(* PLC project Unnamed, Unknown Unnamed 1 *)
(* stored: creationDateTime 2021-10-03T01:48:44, modificationDateTime 2021-10-03T03:04:46 *)

PROGRAM part2
  VAR
    pos_x0 AT %IX0.0 : BOOL;
    pos_x1 AT %IX0.1 : BOOL;
    pos_x2 AT %IX0.2 : BOOL;
    pos_x3 AT %IX0.3 : BOOL;
  END_VAR
  VAR
    pos_x : UINT;
  END_VAR
  VAR
    pos_y0 AT %IX0.4 : BOOL;
    pos_y1 AT %IX0.5 : BOOL;
    pos_y2 AT %IX0.6 : BOOL;
    pos_y3 AT %IX0.7 : BOOL;
    target_x0 AT %IX1.0 : BOOL;
    target_x1 AT %IX1.1 : BOOL;
    target_x2 AT %IX1.2 : BOOL;
    target_x3 AT %IX1.3 : BOOL;
    target_y0 AT %IX1.4 : BOOL;
    target_y1 AT %IX1.5 : BOOL;
    target_y2 AT %IX1.6 : BOOL;
    target_y3 AT %IX1.7 : BOOL;
    dir_up AT %QX0.0 : BOOL;
    dir_down AT %QX0.1 : BOOL;
    dir_left AT %QX0.2 : BOOL;
    dir_right AT %QX0.3 : BOOL;
  END_VAR
  VAR  (* added by the conversion: wires and edge detectors of the diagram *)
    _ADD42_OUT : UINT;
    _ADD31_OUT : UINT;
    _ADD79_OUT : UINT;
    _ADD73_OUT : UINT;
  END_VAR

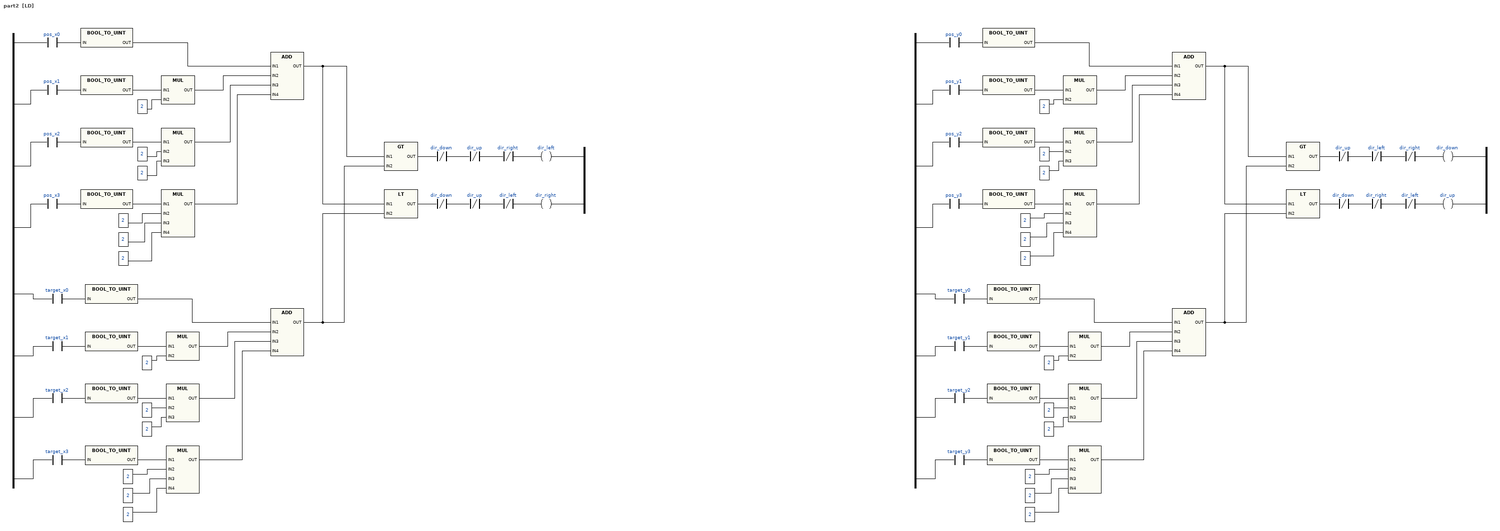
(* LD diagram, written out as Structured Text *)
_ADD42_OUT := BOOL_TO_UINT(pos_x0) + BOOL_TO_UINT(pos_x1) * 2 + BOOL_TO_UINT(pos_x2) * 2 * 2 + BOOL_TO_UINT(pos_x3) * 2 * 2 * 2;
_ADD31_OUT := BOOL_TO_UINT(target_x0) + BOOL_TO_UINT(target_x1) * 2 + BOOL_TO_UINT(target_x2) * 2 * 2 + BOOL_TO_UINT(target_x3) * 2 * 2 * 2;
dir_left := _ADD42_OUT > _ADD31_OUT AND NOT dir_down AND NOT dir_up AND NOT dir_right;
_ADD79_OUT := BOOL_TO_UINT(pos_y0) + BOOL_TO_UINT(pos_y1) * 2 + BOOL_TO_UINT(pos_y2) * 2 * 2 + BOOL_TO_UINT(pos_y3) * 2 * 2 * 2;
_ADD73_OUT := BOOL_TO_UINT(target_y0) + BOOL_TO_UINT(target_y1) * 2 + BOOL_TO_UINT(target_y2) * 2 * 2 + BOOL_TO_UINT(target_y3) * 2 * 2 * 2;
dir_down := _ADD79_OUT > _ADD73_OUT AND NOT dir_up AND NOT dir_left AND NOT dir_right;
dir_right := _ADD42_OUT < _ADD31_OUT AND NOT dir_down AND NOT dir_up AND NOT dir_left;
dir_up := _ADD79_OUT < _ADD73_OUT AND NOT dir_down AND NOT dir_right AND NOT dir_left;
END_PROGRAM

CONFIGURATION Config0
  RESOURCE Res0 ON PLC
    TASK task0(INTERVAL := T#20ms, PRIORITY := 0);
    PROGRAM instance0 WITH task0 : part2;
  END_RESOURCE
END_CONFIGURATION
